FUNCTION Zbm3 : REAL
VAR_INPUT
END_VAR
VAR
END_VAR

END_FUNCTION

(* stored: Version 1.1.0.1, ProductVersion 3.1.4024.6
   POU Zbm3: Id {11fa347d-b7bb-4cbb-b0d1-3f950d382f1a}, SpecialFunc None *)
